// TIA Portal V19 export
TYPE "C701_VAR_IF_VCO_TYPIC"
   STRUCT
      REQ_VE { ExternalAccessible := 'False'; ExternalVisible := 'False'; ExternalWritable := 'False'} : Bool;   // Warmtevraag
      REQ_KO { ExternalAccessible := 'False'; ExternalVisible := 'False'; ExternalWritable := 'False'} : Bool;   // Koelvraag
      TME_HOLA { ExternalAccessible := 'False'; ExternalVisible := 'False'; ExternalWritable := 'False'} : Bool;   // Ruimtetemperatuur te hoog of te laag
      STO { ExternalAccessible := 'False'; ExternalVisible := 'False'; ExternalWritable := 'False'} : Bool;   // Storing algemeen ventiloconvector
   END_STRUCT;
END_TYPE
